PROGRAM PMPS_Arbiter
VAR

	fbSetPE	:	PE_Ranges;

    fbBPRequestor : FB_BPRequestor; // Updates global PMPS RequestedBeamParams
    {attribute 'pytmc' := '
    pv: @(PREFIX)PhotonEnergyWatcher
    '}
    fbPhotonEnergyWatcher	:	FB_PhotonEnergyWatcher;
    {attribute 'pytmc' := '
    pv: @(PREFIX)BeamClassOutputs
    '}
    fbMPSInterface	:	FB_BeamClassOutputs;
    {attribute 'pytmc' := '
    pv: @(PREFIX)CuRateOutputs
    '}
    fbCuInterface	:	FB_CTLS_Outputs;

    (* Subsystem requests use this FB and a pragma link to pass their requests to the arbiter.
    The fb is called on each cycle and updates the arbiter with the current BP set requested
    from the subsystem PLC.*)
    //<TODO> make this so it does input and output to the IF
    (*{attribute 'pytmc' := '
    pv: @(PREFIX):PLC1
    '}*)
    {attribute 'TcLinkTo' := '.i_RequestedBP:=TIIB[plc-kfe-motion]^IO Inputs^RequestedBP;
                                .o_CurrentBP:=TIIB[plc-kfe-motion]^IO Outputs^CurrentBP;
                                .i_Connected:=TIIB[plc-kfe-motion]^SYNC Inputs^External device not connected;
                                .i_WcState:=TIIB[plc-kfe-motion]^WcState^WcStateIn;
                                .i_TxPDOState:=TIIB[plc-kfe-motion]^SYNC Inputs^TxPDO state;
                                '}
    plc_kfe_motion_PMPS_IO : FB_ArbiterToSubSys_IO := (RequestingSystemID := 16#FF0F);
	
	    {attribute 'TcLinkTo' := '.i_RequestedBP:=TIIB[plc-kfe-optics]^IO Inputs^RequestedBP;
                                .o_CurrentBP:=TIIB[plc-kfe-optics]^IO Outputs^CurrentBP;
                                .i_Connected:=TIIB[plc-kfe-optics]^SYNC Inputs^External device not connected;
                                .i_WcState:=TIIB[plc-kfe-optics]^WcState^WcStateIn;
                                .i_TxPDOState:=TIIB[plc-kfe-optics]^SYNC Inputs^TxPDO state;
                                '}
    plc_kfe_optics_PMPS_IO : FB_ArbiterToSubSys_IO := (RequestingSystemID := 16#FF10);

	
	{attribute 'TcLinkTo' := '.i_RequestedBP:=TIIB[plc-kfe-vac]^IO Inputs^RequestedBP;
								.o_CurrentBP:=TIIB[plc-kfe-vac]^IO Outputs^CurrentBP;
								.i_Connected:=TIIB[plc-kfe-vac]^SYNC Inputs^External device not connected;
								.i_WcState:=TIIB[plc-kfe-vac]^WcState^WcStateIn;
								.i_TxPDOState:=TIIB[plc-kfe-vac]^SYNC Inputs^TxPDO state;
								'}
    plc_kfe_vac_PMPS_IO : FB_ArbiterToSubSys_IO := (RequestingSystemID := 16#FF11);
	
	{attribute 'TcLinkTo' := '.i_RequestedBP:=TIIB[plc-kfe-gatt]^IO Inputs^RequestedBP;
								.o_CurrentBP:=TIIB[plc-kfe-gatt]^IO Outputs^CurrentBP;
								.i_Connected:=TIIB[plc-kfe-gatt]^SYNC Inputs^External device not connected;
								.i_WcState:=TIIB[plc-kfe-gatt]^WcState^WcStateIn;
								.i_TxPDOState:=TIIB[plc-kfe-gatt]^SYNC Inputs^TxPDO state;
								'}
    plc_kfe_gatt_PMPS_IO : FB_ArbiterToSubSys_IO := (RequestingSystemID := 16#FF12);
	
	{attribute 'TcLinkTo' := '.i_RequestedBP:=TIIB[plc-kfe-gmd-vac-01]^IO Inputs^RequestedBP;
								.o_CurrentBP:=TIIB[plc-kfe-gmd-vac-01]^IO Outputs^CurrentBP;
								.i_Connected:=TIIB[plc-kfe-gmd-vac-01]^SYNC Inputs^External device not connected;
								.i_WcState:=TIIB[plc-kfe-gmd-vac-01]^WcState^WcStateIn;
								.i_TxPDOState:=TIIB[plc-kfe-gmd-vac-01]^SYNC Inputs^TxPDO state;
								'}
    plc_kfe_gmd_PMPS_IO : FB_ArbiterToSubSys_IO := (RequestingSystemID := 16#FF13);
	
	{attribute 'TcLinkTo' := '.i_RequestedBP:=TIIB[plc-kfe-xgmd-vac-01]^IO Inputs^RequestedBP;
								.o_CurrentBP:=TIIB[plc-kfe-xgmd-vac-01]^IO Outputs^CurrentBP;
								.i_Connected:=TIIB[plc-kfe-xgmd-vac-01]^SYNC Inputs^External device not connected;
								.i_WcState:=TIIB[plc-kfe-xgmd-vac-01]^WcState^WcStateIn;
								.i_TxPDOState:=TIIB[plc-kfe-xgmd-vac-01]^SYNC Inputs^TxPDO state;
								'}
    plc_kfe_xgmd_PMPS_IO : FB_ArbiterToSubSys_IO := (RequestingSystemID := 16#FF14);
	
	
	
	//////////////////////////////////////////////
	// TMO PLCs
	/////////////////////////////////////////////
	
	{attribute 'TcLinkTo' := '.i_RequestedBP:=TIIB[plc-tmo-mot]^IO Inputs^RequestedBP;
                                .o_CurrentBP:=TIIB[plc-tmo-mot]^IO Outputs^CurrentBP;
                                .i_Connected:=TIIB[plc-tmo-mot]^SYNC Inputs^External device not connected;
                                .i_WcState:=TIIB[plc-tmo-mot]^WcState^WcStateIn;
                                .i_TxPDOState:=TIIB[plc-tmo-mot]^SYNC Inputs^TxPDO state;
                                '}
    plc_tmo_motion_PMPS_IO : FB_ArbiterToSubSys_IO := (RequestingSystemID := 16#F100);
	
	{attribute 'TcLinkTo' := '.i_RequestedBP:=TIIB[plc-tmo-optics]^IO Inputs^RequestedBP;
                                .o_CurrentBP:=TIIB[plc-tmo-optics]^IO Outputs^CurrentBP;
                                .i_Connected:=TIIB[plc-tmo-optics]^SYNC Inputs^External device not connected;
                                .i_WcState:=TIIB[plc-tmo-optics]^WcState^WcStateIn;
                                .i_TxPDOState:=TIIB[plc-tmo-optics]^SYNC Inputs^TxPDO state;
                                '}
    plc_tmo_optics_PMPS_IO : FB_ArbiterToSubSys_IO := (RequestingSystemID := 16#F101);

	{attribute 'TcLinkTo' := '.i_RequestedBP:=TIIB[plc-tmo-vac]^IO Inputs^RequestedBP;
                                .o_CurrentBP:=TIIB[plc-tmo-vac]^IO Outputs^CurrentBP;
                                .i_Connected:=TIIB[plc-tmo-vac]^SYNC Inputs^External device not connected;
                                .i_WcState:=TIIB[plc-tmo-vac]^WcState^WcStateIn;
                                .i_TxPDOState:=TIIB[plc-tmo-vac]^SYNC Inputs^TxPDO state;
                                '}
    plc_tmo_vacuum_PMPS_IO : FB_ArbiterToSubSys_IO := (RequestingSystemID := 16#F102);	
	
	count : CTU;

END_VAR


// Updating arbiter with subsystem requests.

///////////////////////////
// KFE
	plc_kfe_motion_PMPS_IO(Arbiter:=GVL.g_fbArbiter1, fbFFHWO:=GVL.g_FastFaultOutput1, Reset:=GVL.AttemptReset);
	plc_kfe_optics_PMPS_IO(Arbiter:=GVL.g_fbArbiter1, fbFFHWO:=GVL.g_FastFaultOutput1, Reset:=GVL.AttemptReset);
	plc_kfe_vac_PMPS_IO(Arbiter:=GVL.g_fbArbiter1, fbFFHWO:=GVL.g_FastFaultOutput1, Reset:=GVL.AttemptReset);
	plc_kfe_gatt_PMPS_IO(Arbiter:=GVL.g_fbArbiter1, fbFFHWO:=GVL.g_FastFaultOutput1, Reset:=GVL.AttemptReset);


///////////////////////////
// TMO
	plc_tmo_motion_PMPS_IO(Arbiter:=GVL.g_fbArbiter1, fbFFHWO:=GVL.g_FastFaultOutput1, Reset:=GVL.AttemptReset);
	plc_tmo_optics_PMPS_IO(Arbiter:=GVL.g_fbArbiter1, fbFFHWO:=GVL.g_FastFaultOutput1, Reset:=GVL.AttemptReset);
	plc_tmo_vacuum_PMPS_IO(Arbiter:=GVL.g_fbArbiter1, fbFFHWO:=GVL.g_FastFaultOutput1, Reset:=GVL.AttemptReset);

	
	
////////////////////////////	
// Beam parameter requestor
fbBPRequestor(Arbiter:=GVL.g_fbArbiter1, q_ReqBP => PMPS_GVL.stRequestedBeamParameters);

// Request beam class
fbMPSInterface(BP := PMPS_GVL.stRequestedBeamParameters);

// Request Cu beam rate
fbCuInterface(BP := PMPS_GVL.stRequestedBeamParameters);


// Keep an eye on the photon energy
fbPhotonEnergyWatcher(i_stCurrentBeamParams	:= PMPS_GVL.stCurrentBeamParameters,
                    i_stRequestedBeamParams := PMPS_GVL.stRequestedBeamParameters,
                    io_fbFFHWO:= GVL.g_FastFaultOutput1,
                    i_xReset := GVL.AttemptReset);			

// Evaluate fast fault vetos
g_FastFaultOutput1.Execute();

END_PROGRAM

(* stored: Version 1.1.0.1, ProductVersion 3.1.4022.18
   POU PMPS_Arbiter: Id {91ae890b-11cc-4d41-83ec-edc5b802c784}, SpecialFunc None *)
